FUNCTION_BLOCK ASM_CTL (* Controller for Simple Assembly Station with Dual-Cylinder Transport *)
  (* Standard: 61499-1; ApplicationDomain: Assembly; Function: Control *)
  (* Version 0.1, 2004-10-21, JHC, Rockwell Automation, Changed a transition from P_HOME to NOT P_END. *)
  (* Version 0.0, 2004-09-25, JHC, Rockwell Automation, Adapted from ASM_CTL. *)
  (* Compiler header: package fb.rt.mach; import fb.rt.math.*; *)
  (* Compiler Java Sun JDK 1.4.2 *)
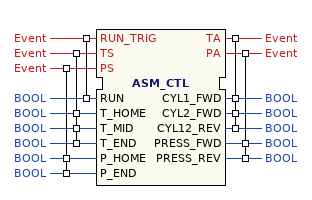
  EVENT_INPUT
    RUN_TRIG WITH RUN; (* RUN/STOP trigger *)
    TS WITH T_HOME, T_MID, T_END; (* Transport Sensors *)
    PS WITH P_HOME, P_END; (* Press Sensors *)
  END_EVENT
  EVENT_OUTPUT
    TA WITH CYL1_FWD, CYL2_FWD, CYL12_REV; (* Transport Actuators *)
    PA WITH PRESS_REV, PRESS_FWD; (* Press Actuators *)
  END_EVENT
  VAR_INPUT
    RUN : BOOL; (* Enable cycling *)
    T_HOME : BOOL; (* Transport at HOME position *)
    T_MID : BOOL; (* Transport at MID position *)
    T_END : BOOL; (* Transport at END position *)
    P_HOME : BOOL; (* Press at HOME position *)
    P_END : BOOL; (* Press at END position *)
  END_VAR
  VAR_OUTPUT
    CYL1_FWD : BOOL; (* Move Cylinder#1 Forward *)
    CYL2_FWD : BOOL; (* Move Cylinder#2 Forward *)
    CYL12_REV : BOOL; (* Retract Both Cylinders *)
    PRESS_FWD : BOOL; (* Move Press Forward *)
    PRESS_REV : BOOL; (* Retract Press *)
  END_VAR
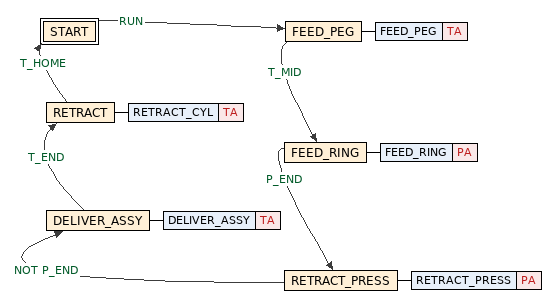
  EC_STATES
    START; (* Initial State *)
    FEED_PEG : FEED_PEG -> TA;
    FEED_RING : FEED_RING -> PA;
    RETRACT_PRESS : RETRACT_PRESS -> PA;
    DELIVER_ASSY : DELIVER_ASSY -> TA;
    RETRACT : RETRACT_CYL -> TA;
  END_STATES
  EC_TRANSITIONS
    START TO FEED_PEG := RUN;
    FEED_PEG TO FEED_RING := T_MID;
    FEED_RING TO RETRACT_PRESS := P_END;
    RETRACT_PRESS TO DELIVER_ASSY := NOT P_END;
    DELIVER_ASSY TO RETRACT := T_END;
    RETRACT TO START := T_HOME;
  END_TRANSITIONS
  ALGORITHM FEED_PEG IN ST:
CYL1_FWD := TRUE;
CYL2_FWD := FALSE;
CYL12_REV := FALSE;
  END_ALGORITHM
  ALGORITHM FEED_RING IN ST:
PRESS_FWD := TRUE;
PRESS_REV := FALSE;
  END_ALGORITHM
  ALGORITHM RETRACT_PRESS IN ST:
PRESS_FWD := FALSE;
PRESS_REV := TRUE;
  END_ALGORITHM
  ALGORITHM DELIVER_ASSY IN ST:
CYL1_FWD := TRUE;
CYL2_FWD := TRUE;
CYL12_REV := FALSE;
  END_ALGORITHM
  ALGORITHM RETRACT_CYL IN ST:
CYL1_FWD := FALSE;
CYL2_FWD := FALSE;
CYL12_REV := TRUE;
  END_ALGORITHM
END_FUNCTION_BLOCK
